# EPICS IOC start-up script: isrc-010_ctrl-plc-01.cmd-test-20191106135317.iocsh
# @field isrc-010_ctrl-plc-01_VERSION
# @runtime YES

# Load plc interface database
dbLoadRecords("isrc-010_ctrl-plc-01-test.db", "MODVERSION=$(isrc-010_ctrl-plc-01_VERSION)")
